Fanuc TP program (LS listing): message14.ls

/PROG  MESSAGE14	  Macro
/ATTR
OWNER		= MNEDITOR;
COMMENT		= "USER MESSAGE";
PROG_SIZE	= 283;
CREATE		= DATE 22-05-16  TIME 15:52:26;
MODIFIED	= DATE 22-05-17  TIME 09:34:26;
FILE_NAME	= MESSAGE1;
VERSION		= 0;
LINE_COUNT	= 2;
MEMORY_SIZE	= 663;
PROTECT		= READ_WRITE;
TCD:  STACK_SIZE	= 0,
      TASK_PRIORITY	= 50,
      TIME_SLICE	= 0,
      BUSY_LAMP_OFF	= 0,
      ABORT_REQUEST	= 0,
      PAUSE_REQUEST	= 7;
DEFAULT_GROUP	= *,*,*,*,*;
CONTROL_CODE	= 00000000 00000000;
/APPL
/APPL

AUTO_SINGULARITY_HEADER;
  ENABLE_SINGULARITY_AVOIDANCE   : FALSE;
/MN
   1:  CALL MESSAGE20    ;
   2:  CALL FAULT_MESSAGE('A side pallet setup complete.') ;
/POS
/END
